{attribute 'Tc2GvlVarNames'}
VAR_GLOBAL

	bAutoSysOn			: BOOL;
	bSevenDaySysOn 	: BOOL;
	bSevenDaySysOff 	: BOOL;

END_VAR

(* stored: Version 1.1.0.1, ProductVersion 3.1.4024.12
   GVL Global_Variables_SevenDay_NoPersistent: Id {075a852e-e20f-4e90-aa49-7f6977e97226} *)
